// TIA Portal V19 export
TYPE "ValveMachine_COut"
// stored: Access Published
   STRUCT
      CtrlSafe : Bool;
      Standstill : Bool;
      ReqOilPressure : Bool;
      Rest_CheckNext : Bool;   // Move to rest position requested
      Work_CheckNext : Bool;   // Move to work position requested
      Rest : Bool;   // Actuator is in rest position
      Work : Bool;   // Actuator is in work position
   END_STRUCT;
END_TYPE
